// TIA Portal project "FactoryIO_Template_S7-1200_V15_V15.1" (V15.1)
// Vorlageprojekt für das Buch mit Zielsystem S7-1200

(* hardware
DEVICE "S7-1200-Station_1"  S7-1200 Station
   slot 0: "Baugruppenträger_0"  Rack  V1.0
   slot 1: "PLC_1"  CPU 1211C DC/DC/DC  6ES7 211-1AE40-0XB0  V4.1
*)

// ===== PLC "PLC_1"  CPU 1211C DC/DC/DC =====

VAR_GLOBAL   // PLC tag table "Standard-Variablentabelle"
   "Conveyor" AT %A0.0 : Bool;
   "Sensor A" AT %E0.0 : Bool;
   "Sensor B" AT %E0.1 : Bool;
   "LED_A" AT %Q0.1 : Bool;
   "LED_B" AT %Q0.2 : Bool;
   "Entry_Conveyor" AT %Q0.3 : Bool;
END_VAR

DATA_BLOCK "Auxiliare"   // DB1
{ S7_Optimized_Access := 'TRUE' }
VERSION : 0.1
   VAR
      trecut_A : Bool;
   END_VAR
BEGIN
END_DATA_BLOCK

FUNCTION "MHJ-PLC-Lab-Function-S71200" : Void   // FC9000, SCL
{ S7_Optimized_Access := 'TRUE' }
VERSION : 0.1
   VAR_TEMP
      rdTimeReturn : Int;
      outputTime : DTL;
      SyncVal : Byte;
      forVal : Int;
      forVal_2 : Int;
      Value : Byte;
   END_VAR
   VAR CONSTANT
      CompVal : Byte := 16#34;
      Value_01 : Byte := 16#11;
      Value_01_DW : DWord := 16#A165_D992;
      Value_02_DW : DWord := 16#58BE_4401;
   END_VAR
BEGIN

   #Value:=PEEK(area := 16#82,
        dbNumber := 0,
        byteOffset := 511);
   #Value := #Value + 1;

   POKE(area := 16#82,
        dbNumber := 0,
        byteOffset := 511,
        value := #Value);

   POKE(area:=16#81,
        dbNumber:=0,
        byteOffset:=1016,
        value:=#Value_01_DW);
   POKE(area := 16#81,
        dbNumber := 0,
        byteOffset := 1020,
        value := #Value_02_DW);

   POKE(area := 16#81,
        dbNumber := 0,
        byteOffset := 511,
        value := B#16#00);

   FOR #forVal := 0 TO 120 DO
       FOR #forVal_2:=0 TO 10 DO
           #rdTimeReturn:=RD_SYS_T(#outputTime);
           #rdTimeReturn := WR_SYS_T(#outputTime);
           #rdTimeReturn := RD_SYS_T(#outputTime);
           #rdTimeReturn := WR_SYS_T(#outputTime);
       END_FOR;
       #SyncVal:= PEEK(area := 16#81,
                      dbNumber := 0,
                      byteOffset := 511);
       IF #SyncVal = #CompVal THEN
          GOTO M_1;
       END_IF;
   END_FOR;
   RETURN;

   M_1:
   POKE(area := 16#81,
        dbNumber := 0,
        byteOffset := 511,
        value := B#16#0);
END_FUNCTION

ORGANIZATION_BLOCK "Main"   // OB1, LAD, ProgramCycle
TITLE = "Main Program Sweep (Cycle)"
{ S7_Optimized_Access := 'TRUE' }
VERSION : 0.1
   VAR_INPUT
      Initial_Call : Bool;   // Initial call of this OB
      Remanence : Bool;   // =True, if remanent data are available
   END_VAR
BEGIN

REGION Network 1: Konnektierungsbaustein für PLC-Lab
   // Im Netzwerk 1 wird der Konnektierungsbaustein für PLC-Lab aufgerufen.
   // Dieser Aufruf darf nicht entfernt werden!
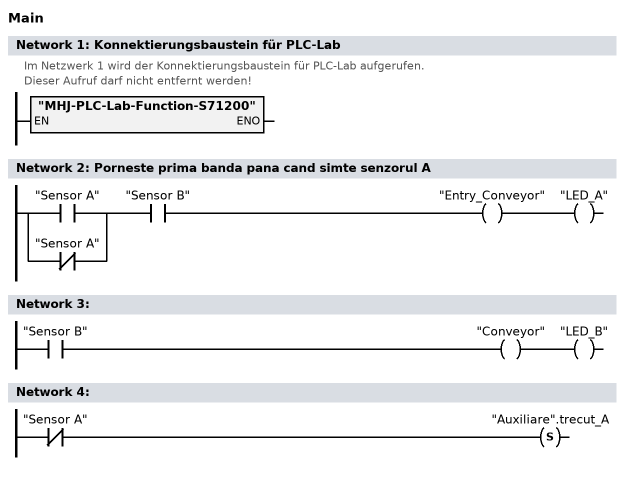
   RUNG wire#powerrail
      "MHJ-PLC-Lab-Function-S71200"()
   END_RUNG
   // the same network as SCL:
   "MHJ-PLC-Lab-Function-S71200"();
END_REGION

REGION Network 2: Porneste prima banda pana cand simte senzorul A
   RUNG wire#powerrail
      Contact( "Sensor A" )
      wire#w1
      Contact( "Sensor B" )
      Coil( "Entry_Conveyor" )
      Coil( "LED_A" )
   END_RUNG
   RUNG wire#powerrail
      I_Contact( "Sensor A" )
   END_RUNG wire#w1
   // the same network as SCL:
   "Entry_Conveyor" := ("Sensor A" OR NOT "Sensor A") AND "Sensor B";
   "LED_A" := "Entry_Conveyor";
END_REGION

REGION Network 3
   RUNG wire#powerrail
      Contact( "Sensor B" )
      Coil( "Conveyor" )
      Coil( "LED_B" )
   END_RUNG
   // the same network as SCL:
   "Conveyor" := "Sensor B";
   "LED_B" := "Sensor B";
END_REGION

REGION Network 4
   RUNG wire#powerrail
      I_Contact( "Sensor A" )
      S_Coil( "Auxiliare".trecut_A )
   END_RUNG
   // the same network as SCL:
   IF NOT "Sensor A" THEN "Auxiliare".trecut_A := TRUE; END_IF;
END_REGION
END_ORGANIZATION_BLOCK